// TIA Portal V20 export
TYPE "typeEmDataControlNode"
// stored: Namespace Unit1.Em5
   STRUCT
      sideTape : "LER_typePartData";
      hotPressLeft { S7_SetPoint := 'True'} : "LER_typePartData";
      hotPressRight { S7_SetPoint := 'True'} : "LER_typePartData";
      transferPnPLeft : "LER_typePartData";
      transferPnPRight : "LER_typePartData";
      hipotThickness : "LER_typePartData";
      vision : "LER_typePartData";
      laserMark : "LER_typePartData";
   END_STRUCT;
END_TYPE
